// Mitsubishi GX Works2 project: LRI - PLC - OR   PLC: Q03UDV

PROGRAM MAIN
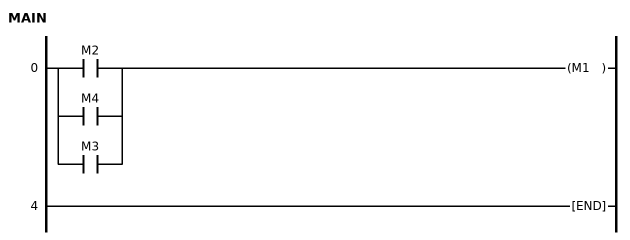
0     LD      M2
      OR      M4
      OR      M3
      OUT     M1
4     END
END_PROGRAM
